TYPE st_EasyPump :
STRUCT
 iPumpType:INT;//泵头类型
 iHosePipeType:INT;//软管类型
END_STRUCT
END_TYPE

(* stored: Version 1.1.0.1, ProductVersion 3.1.4024.9
   DUT st_EasyPump: Id {8bf84668-2b6c-4155-81ca-3fed971bc40c} *)
